Staubli VAL3: init.pgx

public program init(num x_nDetNum, string x_sTask)
  local num l_i
begin
  //***** Customizable section
  //
  //***** end of customizable section
  // ************************
  // do not change anything beyond this line
  //
  //***************************
  //********* Strings *********
  //***************************
  sTASK=x_sTask+toString("",x_nDetNum)
  sDetNum="DET"+toString("",x_nDetNum)
  //
  //***************************
  //*****   Numerics     ******
  //***************************
  // Number of detected objects
  nNumOfPart=-1
  //
  // Resize buffers
  resize(nObjectID,1,nMaxNumOfObject)
  resize(nLatchedValue,1,nMaxNumOfObject)
  resize(trObjectPos,1,nMaxNumOfObject)
  //
  // Initialize ID buffer
  for l_i=0 to size(nObjectID)-1
    nObjectID[l_i]=-1
  endFor
  //
  // Initialize Latched Encoder Value buffer
  for l_i=0 to size(nLatchedValue)-1
    nLatchedValue[l_i]=0
  endFor
  //
  // Initialize TRSF buffer
  for l_i=0 to size(trObjectPos)-1
    trObjectPos[l_i]={0,0,0,0,0,0}
  endFor
  //
  //***************************
  //*****   Booleans     ******
  //***************************
  // Detection library in calibration mode.
  //  Only used by the detection library "Socket".
  bCalibrating=false
  //
end
